(* PLC project WAMPTest, Beremiz Beremiz 1 *)
(* stored: creationDateTime 2015-02-05T11:44:55, modificationDateTime 2020-06-09T10:56:09 *)

PROGRAM program0
  VAR
    LocalVar0 : DINT := 1;
  END_VAR
  VAR_EXTERNAL
    PyVar0 : DINT;
    PyVar1 : DINT;
  END_VAR

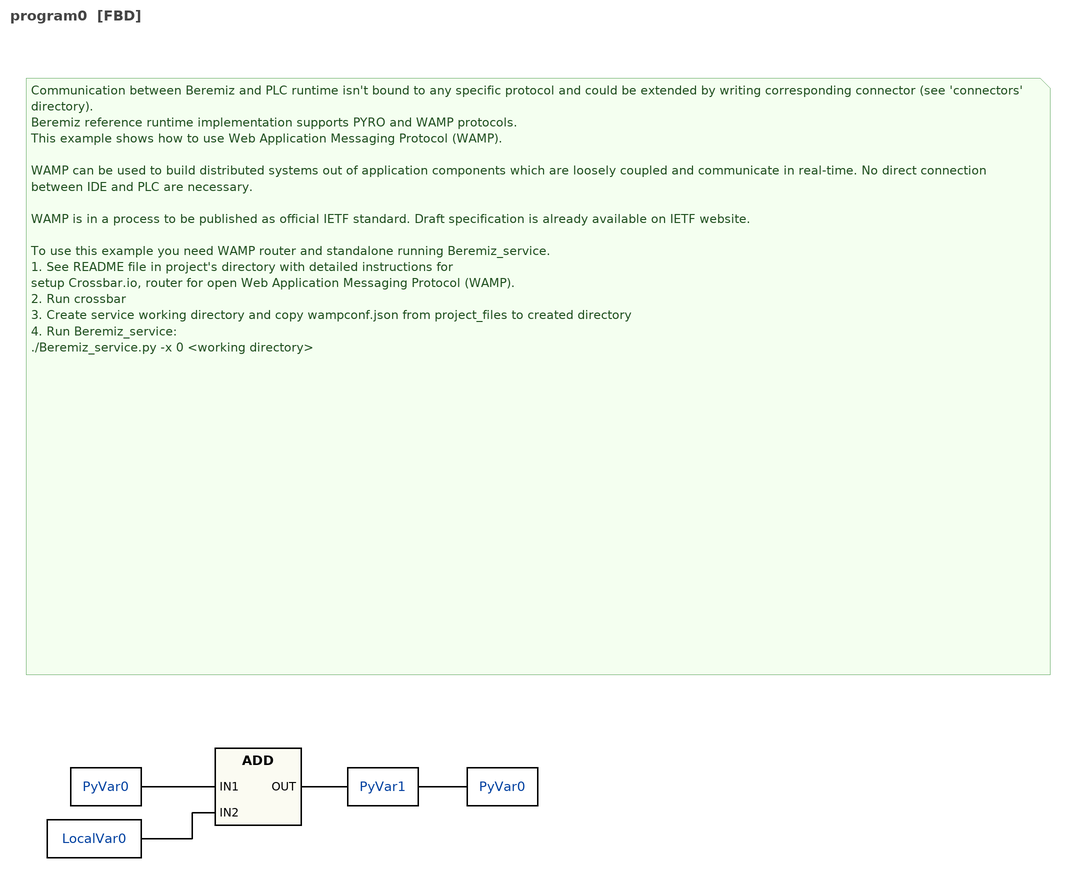
(* FBD diagram, written out as Structured Text *)
(* Communication between Beremiz and PLC runtime isn't bound to any specific protocol and could be extended by writing corresponding connector (see 'connectors' directory).
Beremiz reference runtime implementation supports PYRO and WAMP protocols.
This example shows how to use Web Application Messaging Protocol (WAMP).

WAMP can be used to build distributed systems out of application components which are loosely coupled and communicate in real-time. No direct connection between IDE and PLC are necessary.

WAMP is in a process to be published as official IETF standard. Draft specification is already available on IETF website.
	
To use this example you need WAMP router and standalone running Beremiz_service.
1. See README file in project's directory with detailed instructions for
setup Crossbar.io, router for open Web Application Messaging Protocol (WAMP).
2. Run crossbar
3. Create service working directory and copy wampconf.json from project_files to created directory
4. Run Beremiz_service:
./Beremiz_service.py -x 0 <working directory> *)
PyVar1 := PyVar0 + LocalVar0;
PyVar0 := PyVar1;
END_PROGRAM

CONFIGURATION config
  RESOURCE resource1 ON PLC
    TASK Task0(INTERVAL := T#100ms, PRIORITY := 0);
    PROGRAM Instance0 WITH Task0 : program0;
  END_RESOURCE
END_CONFIGURATION
